SUBAPPLICATION Uebung_002b2 (* DigitalInput_I1/_I2 auf DigitalOutput_Q1 *)
  (* Standard: 61499-2 *)
  (* Version 1.0, 2023-10-23, franz *)
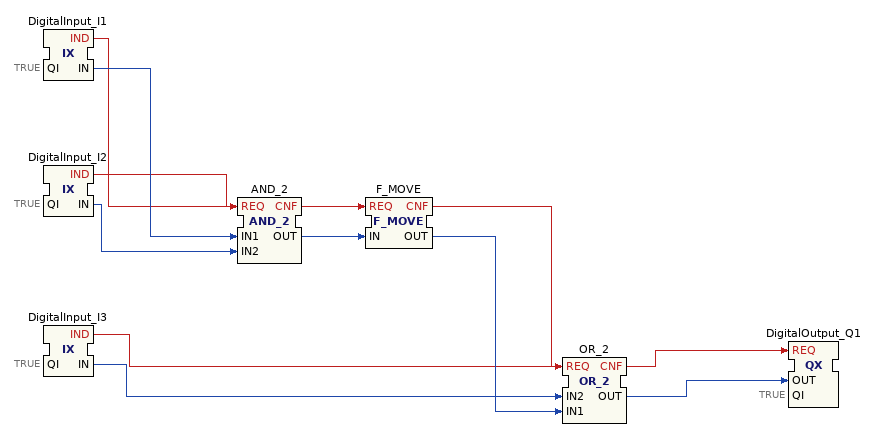
  FBS
    DigitalOutput_Q1 : QX(QI := TRUE);
    DigitalInput_I1 : IX(QI := TRUE);
    DigitalInput_I2 : IX(QI := TRUE);
    AND_2 : AND_2;
    DigitalInput_I3 : IX(QI := TRUE);
    OR_2 : OR_2;
    F_MOVE : F_MOVE; {SET_ATTRIBUTE(DataType, BOOL)}
  END_FBS
  EVENT_CONNECTIONS
    DigitalInput_I1.IND TO AND_2.REQ;
    DigitalInput_I2.IND TO AND_2.REQ;
    OR_2.CNF TO DigitalOutput_Q1.REQ;
    DigitalInput_I3.IND TO OR_2.REQ;
    AND_2.CNF TO F_MOVE.REQ;
    F_MOVE.CNF TO OR_2.REQ;
  END_CONNECTIONS
  DATA_CONNECTIONS
    DigitalInput_I1.IN TO AND_2.IN1;
    DigitalInput_I2.IN TO AND_2.IN2;
    DigitalInput_I3.IN TO OR_2.IN2;
    OR_2.OUT TO DigitalOutput_Q1.OUT;
    AND_2.OUT TO F_MOVE.IN;
    F_MOVE.OUT TO OR_2.IN1;
  END_CONNECTIONS
END_SUBAPPLICATION
